FUNCTION_BLOCK FB_SlitPairV2
VAR_INPUT
    nIdPositiveAxis: UINT; //ID of axis for which positive motion increases gap size
    nIdNegativeAxis: UINT; //ID of axis for which negative motion increases gap size
    nIdGapSizeAxis: UINT; //ID of virtual gap aperture size axis
    nIdGapCentreAxis: UINT; //ID of virtual gap centre position axis

    bEnable: BOOL; //Enable slit pair logic functionality
    bReset: BOOL; //Reset from error state
    fEncoderScaling: LREAL := 10000; //Virtual axis scaling denominator, default of 10000
END_VAR
VAR
    nGapSizeEncoder AT %Q*: UDINT := 0;
    nGapCentreEncoder AT %Q*: UDINT := 0;
    fGapSize: LREAL;
    fGapCentre: LREAL;
    bAllHalted: BOOL := FALSE;
    bInternalResetHome: BOOL :=FALSE;

    fbSetpointGenEnablePositiveAxis: MC_ExtSetPointGenEnable;
    fbSetpointGenEnableNegativeAxis: MC_ExtSetPointGenEnable;
    fbSetpointGenEnableGapSizeAxis: MC_ExtSetPointGenEnable;
    fbSetpointGenEnableGapCentreAxis: MC_ExtSetPointGenEnable;

    fbSetpointGenDisablePositiveAxis: MC_ExtSetPointGenDisable;
    fbSetpointGenDisableNegativeAxis: MC_ExtSetPointGenDisable;
    fbSetpointGenDisableGapSizeAxis: MC_ExtSetPointGenDisable;
    fbSetpointGenDisableGapCentreAxis: MC_ExtSetPointGenDisable;

    fPosSetpointPositiveAxis: LREAL;
    fPosSetpointNegativeAxis: LREAL;
    fPosSetpointGapSizeAxis: LREAL;
    fPosSetpointGapCentreAxis: LREAL;

    fVeloSetpointPositiveAxis: LREAL;
    fVeloSetpointNegativeAxis: LREAL;
    fVeloSetpointGapSizeAxis: LREAL;
    fVeloSetpointGapCentreAxis: LREAL;

    nDirectionPositiveAxis: DINT;
    nDirectionNegativeAxis: DINT;
    nDirectionGapSizeAxis: DINT;
    nDirectionGapCentreAxis: DINT;

    eState: E_SlitPairStatesV2 := E_SlitPairStatesV2.eInit;

    bInternalReset: BOOL;
    bHomingReset: BOOL := FALSE;

    //Two resets required due to homing functionality
    bResetInProgressCheck1: BOOL := FALSE;
    bResetInProgressCheck2: BOOL := FALSE;

    //internal MCPOWER blocks because Beckhoff won't let you enable a setpoint generator on a limit....
    fbPowerPositiveAxis: MC_POWER;
    fbPowerNegativeAxis: MC_POWER;
    fbPowerGapSizeAxis: MC_POWER;
    fbPowerGapCentreAxis: MC_POWER;

    //internal MC_Reset, needed because the current reset in FB_Axis works only when there is an error. This should change once the reset functionality changes
    fbInternalResetTrig: R_TRIG;
    fbInternalResetHome: R_TRIG;
    fbResetPositiveAxis: MC_RESET;
    fbResetNegativeAxis: MC_RESET;
    fbResetGapSizeAxis: MC_RESET;
    fbResetGapCentreAxis: MC_RESET;
    fbResetHomedGap: MC_Home;
    fbResetHomedCentre: MC_Home;

END_VAR


(*SETUP INSTRUCTIONS
Virtual axes:
Encoder type set to Universal
Encoder mask set to 0xFFFFFFFF
Encoder scaling set to match FB
Link nDataIn1 of encoder to FB encoders
Position lag monitoring can be left on*
Dynamics of virtual axes must be configured considering coupled mechanicals (e.g. don't set velocities your real axes can't achieve)
*)

//Position of virtual axes
actVirtualAxisPositions();
//Limit logic
actVirtualAxisLimits();
//Enable Logic - Virtual axes automatically enable when real axes are enabled
actVirtualAxisEnable();
//Call spGenerator FBs
actGeneratorEnableDisable();
//Calculate position setpoints
actCalculateSetpointPositions();
//Calculate velocity setpoints
actCalculateSetpointVelocities();
//Calculate directions
actCalculateSetpointDirections();

//Error state handling - only handle errors that disable motion
IF bEnable AND (GVL.astAxesLocal[nIdPositiveAxis].Axis.Status.ErrorStop OR GVL.astAxesLocal[nIdNegativeAxis].Axis.Status.ErrorStop OR GVL.astAxesLocal[nIdGapSizeAxis].Axis.Status.ErrorStop OR GVL.astAxesLocal[nIdGapCentreAxis].Axis.Status.ErrorStop) THEN
    eState := E_SlitPairStatesV2.eError;
END_IF

//Propagate real axis error to virtual
IF GVL.astAxesLocal[nIdPositiveAxis].Axis.Status.ErrorStop AND (NOT GVL.astAxesLocal[nIdGapSizeAxis].Axis.Status.ErrorStop OR NOT GVL.astAxesLocal[nIdGapCentreAxis].Axis.Status.ErrorStop) THEN
    GVL.astAxesLocal[nIdGapSizeAxis].stStatus.bError := TRUE;
    GVL.astAxesLocal[nIdGapCentreAxis].stStatus.bError := TRUE;
    GVL.astAxesLocal[nIdGapSizeAxis].stStatus.nErrorID := GVL.astAxesLocal[nIdPositiveAxis].stStatus.nErrorID;
    GVL.astAxesLocal[nIdGapCentreAxis].stStatus.nErrorID := GVL.astAxesLocal[nIdPositiveAxis].stStatus.nErrorID;
ELSIF  GVL.astAxesLocal[nIdNegativeAxis].Axis.Status.ErrorStop AND (NOT GVL.astAxesLocal[nIdGapSizeAxis].Axis.Status.ErrorStop OR NOT GVL.astAxesLocal[nIdGapCentreAxis].Axis.Status.ErrorStop) THEN
    GVL.astAxesLocal[nIdGapSizeAxis].stStatus.bError := TRUE;
    GVL.astAxesLocal[nIdGapCentreAxis].stStatus.bError := TRUE;
    GVL.astAxesLocal[nIdGapSizeAxis].stStatus.nErrorID := GVL.astAxesLocal[nIdNegativeAxis].stStatus.nErrorID;
    GVL.astAxesLocal[nIdGapCentreAxis].stStatus.nErrorID := GVL.astAxesLocal[nIdNegativeAxis].stStatus.nErrorID;
END_IF

//Internal Reset linked to any axis reset
bInternalReset := bReset OR GVL.astAxesLocal[nIdPositiveAxis].stControl.bReset OR GVL.astAxesLocal[nIdNegativeAxis].stControl.bReset OR GVL.astAxesLocal[nIdGapSizeAxis].stControl.bReset OR GVL.astAxesLocal[nIdGapCentreAxis].stControl.bReset;

//If real axis is homing, change state
IF bEnable AND (GVL.astAxesLocal[nIdPositiveAxis].Axis.Status.HomingBusy OR GVL.astAxesLocal[nIdNegativeAxis].Axis.Status.HomingBusy) THEN
    eState := E_SlitPairStatesV2.eWaitForRealHomed;
END_IF

//Link all halt buttons in motors
IF GVL.astAxesLocal[nIdPositiveAxis].stControl.bHalt OR GVL.astAxesLocal[nIdNegativeAxis].stControl.bHalt OR
    GVL.astAxesLocal[nIdGapSizeAxis].stControl.bHalt OR GVL.astAxesLocal[nIdGapCentreAxis].stControl.bHalt THEN
    actHaltAllAxes();
END_IF

//Propagate homing status
fbResetHomedGap(Axis:= GVL.astAxesLocal[nIdGapSizeAxis].Axis, HomingMode:= MC_ResetCalibration);
fbResetHomedCentre(Axis:= GVL.astAxesLocal[nIdGapCentreAxis].Axis, HomingMode:= MC_ResetCalibration);
fbInternalResetHome(CLK:= fbResetHomedCentre.Done OR fbResetHomedGap.Done );
IF NOT GVL.astAxesLocal[nIdPositiveAxis].stStatus.bHomed OR NOT GVL.astAxesLocal[nIdNegativeAxis].stStatus.bHomed THEN
        fbResetHomedGap.Execute := TRUE;
        fbResetHomedCentre.Execute := TRUE;
END_IF

IF fbInternalResetHome.Q THEN
        fbResetHomedGap.Execute := FALSE;
        fbResetHomedCentre.Execute := FALSE;
END_IF


//State machine
IF bEnable THEN
    CASE eState OF  //HOMING LOOP ISSUE
        E_SlitPairStatesV2.eInit:
            //If real axes are calibrated, then home the virtual axes, else go Operatioanl
            fbResetPositiveAxis(Axis:=GVL.astAxesLocal[nIdPositiveAxis].Axis, Execute:=FALSE);
            fbResetNegativeAxis(Axis:=GVL.astAxesLocal[nIdNegativeAxis].Axis, Execute:=FALSE);
            fbResetGapSizeAxis(Axis:=GVL.astAxesLocal[nIdGapSizeAxis].Axis, Execute:=FALSE);
            fbResetGapCentreAxis(Axis:=GVL.astAxesLocal[nIdGapCentreAxis].Axis, Execute:=FALSE);
            IF GVL.astAxesLocal[nIdPositiveAxis].stStatus.bHomed AND GVL.astAxesLocal[nIdNegativeAxis].stStatus.bHomed THEN
               GVL.astAxesLocal[nIdGapSizeAxis].stConfig.eHomeSeq := E_HomingRoutines.eHomeDirect;
               GVL.astAxesLocal[nIdGapCentreAxis].stConfig.eHomeSeq := E_HomingRoutines.eHomeDirect;
               GVL.astAxesLocal[nIdGapSizeAxis].stConfig.fHomePosition := fGapSize;
               GVL.astAxesLocal[nIdGapCentreAxis].stConfig.fHomePosition := fGapCentre;
                eState := E_SlitPairStatesV2.eWaitForVirtualHomed;
            ELSE
                eState := E_SlitPairStatesV2.eOperational;
            END_IF

        E_SlitPairStatesV2.eWaitForVirtualHomed:
            //Wait for virtual axis homing to complete/
            GVL.astAxesLocal[nIdGapSizeAxis].stControl.eCommand := E_MotionFunctions.eHome;
            GVL.astAxesLocal[nIdGapSizeAxis].stControl.bExecute := TRUE;
            GVL.astAxesLocal[nIdGapCentreAxis].stControl.eCommand := E_MotionFunctions.eHome;
            GVL.astAxesLocal[nIdGapCentreAxis].stControl.bExecute := TRUE;
            IF GVL.astAxesLocal[nIdGapSizeAxis].stStatus.bHomed AND GVL.astAxesLocal[nIdGapCentreAxis].stStatus.bHomed THEN
                eState := E_SlitPairStatesV2.eOperational;
            END_IF
            //IF NOT IN HOMING STATE

        E_SlitPairStatesV2.eOperational:
            bResetInProgressCheck1 := FALSE;
            //Detect whether real or virtual axes are moving
            IF GVL.astAxesLocal[nIdGapSizeAxis].stStatus.bMoving OR GVL.astAxesLocal[nIdGapCentreAxis].stStatus.bMoving THEN
                eState := E_SlitPairStatesV2.eEnableRealGenerators;
            END_IF
            IF GVL.astAxesLocal[nIdPositiveAxis].stStatus.bMoving OR GVL.astAxesLocal[nIdNegativeAxis].stStatus.bMoving THEN
                eState := E_SlitPairStatesV2.eEnableVirtualGenerators;
            END_IF

        E_SlitPairStatesV2.eEnableRealGenerators:
            //Hold MC_Power on until generators have enabled
            fbPowerPositiveAxis(Axis:=GVL.astAxesLocal[nIdPositiveAxis].Axis, Enable:=TRUE, Enable_Positive:=TRUE,Enable_Negative:=TRUE);
            fbPowerNegativeAxis(Axis:=GVL.astAxesLocal[nIdNegativeAxis].Axis, Enable:=TRUE, Enable_Positive:=TRUE,Enable_Negative:=TRUE);
            fbSetpointGenEnablePositiveAxis.Execute := TRUE;
            fbSetpointGenEnableNegativeAxis.Execute := TRUE;
            eState := E_SlitPairStatesV2.eCheckRealAxisGeneratorsEnabled;

        E_SlitPairStatesV2.eCheckRealAxisGeneratorsEnabled:
            //Hold MC_Power on until generators have enabled
            fbPowerPositiveAxis(Axis:=GVL.astAxesLocal[nIdPositiveAxis].Axis, Enable:=TRUE, Enable_Positive:=TRUE,Enable_Negative:=TRUE);
            fbPowerNegativeAxis(Axis:=GVL.astAxesLocal[nIdNegativeAxis].Axis, Enable:=TRUE, Enable_Positive:=TRUE,Enable_Negative:=TRUE);
            IF fbSetpointGenEnablePositiveAxis.Enabled AND fbSetpointGenEnableNegativeAxis.Enabled THEN
                eState := E_SlitPairStatesV2.eWaitForVirtualMoveDone;
            END_IF

        E_SlitPairStatesV2.eWaitForVirtualMoveDone:
            IF NOT(GVL.astAxesLocal[nIdGapSizeAxis].stStatus.bMoving OR GVL.astAxesLocal[nIdGapCentreAxis].stStatus.bMoving) THEN
                eState := E_SlitPairStatesV2.eDisableRealGenerators;
            END_IF

        E_SlitPairStatesV2.eDisableRealGenerators:
            fbSetpointGenDisablePositiveAxis.Execute := TRUE;
            fbSetpointGenDisableNegativeAxis.Execute := TRUE;
            eState := E_SlitPairStatesV2.eOperational;

        E_SlitPairStatesV2.eEnableVirtualGenerators:
            //Hold MC_Power on until generators have enabled
            fbPowerGapSizeAxis(Axis:=GVL.astAxesLocal[nIdGapSizeAxis].Axis, Enable:=TRUE, Enable_Positive:=TRUE,Enable_Negative:=TRUE);
            fbPowerGapCentreAxis(Axis:=GVL.astAxesLocal[nIdGapCentreAxis].Axis, Enable:=TRUE, Enable_Positive:=TRUE,Enable_Negative:=TRUE);
            fbSetpointGenEnableGapSizeAxis.Execute := TRUE;
            fbSetpointGenEnableGapCentreAxis.Execute := TRUE;
            eState := E_SlitPairStatesV2.eCheckVirtualAxisGeneratorsEnabled;

        E_SlitPairStatesV2.eCheckVirtualAxisGeneratorsEnabled:
            //Hold MC_Power on until generators have enabled
            fbPowerGapSizeAxis(Axis:=GVL.astAxesLocal[nIdGapSizeAxis].Axis, Enable:=TRUE, Enable_Positive:=TRUE,Enable_Negative:=TRUE);
            fbPowerGapCentreAxis(Axis:=GVL.astAxesLocal[nIdGapCentreAxis].Axis, Enable:=TRUE, Enable_Positive:=TRUE,Enable_Negative:=TRUE);
            IF fbSetpointGenEnableGapSizeAxis.Enabled AND fbSetpointGenEnableGapCentreAxis.Enabled THEN
                eState := E_SlitPairStatesV2.eWaitForRealMoveDone;
            END_IF

        E_SlitPairStatesV2.eWaitForRealMoveDone:
            IF NOT(GVL.astAxesLocal[nIdPositiveAxis].stStatus.bMoving OR GVL.astAxesLocal[nIdNegativeAxis].stStatus.bMoving) THEN
                eState := E_SlitPairStatesV2.eDisableVirtualGenerators;
            END_IF

        E_SlitPairStatesV2.eDisableVirtualGenerators:
            fbSetpointGenDisableGapSizeAxis.Execute := TRUE;
            fbSetpointGenDisableGapCentreAxis.Execute := TRUE;
            eState := E_SlitPairStatesV2.eOperational;

        E_SlitPairStatesV2.eError:
            actHaltAllAxes();

            IF bHomingReset THEN
                bInternalReset := TRUE;
                bResetInProgressCheck1 := TRUE;
                bResetInProgressCheck2 := TRUE;
                bHomingReset := FALSE;
            END_IF
            IF bInternalReset OR bReset OR bResetInProgressCheck2 THEN
                fbResetPositiveAxis(Axis:=GVL.astAxesLocal[nIdPositiveAxis].Axis, Execute:=TRUE);
                fbResetNegativeAxis(Axis:=GVL.astAxesLocal[nIdNegativeAxis].Axis, Execute:=TRUE);
                fbResetGapSizeAxis(Axis:=GVL.astAxesLocal[nIdGapSizeAxis].Axis, Execute:=TRUE);
                fbResetGapCentreAxis(Axis:=GVL.astAxesLocal[nIdGapCentreAxis].Axis, Execute:=TRUE);
                GVL.astAxesLocal[nIdPositiveAxis].stControl.bReset := TRUE;
                GVL.astAxesLocal[nIdNegativeAxis].stControl.bReset := TRUE;
                GVL.astAxesLocal[nIdGapSizeAxis].stControl.bReset := TRUE;
                GVL.astAxesLocal[nIdGapCentreAxis].stControl.bReset := TRUE;
                IF NOT(bResetInProgressCheck1) THEN
                    bResetInProgressCheck2 := FALSE;
                END_IF
            END_IF

            IF NOT(GVL.astAxesLocal[nIdPositiveAxis].stStatus.bError) AND NOT(GVL.astAxesLocal[nIdNegativeAxis].stStatus.bError) AND NOT(GVL.astAxesLocal[nIdGapSizeAxis].stStatus.bError) AND NOT(GVL.astAxesLocal[nIdGapCentreAxis].stStatus.bError) THEN
                eState := E_SlitPairStatesV2.eInit;
            END_IF

        E_SlitPairStatesV2.eWaitForRealHomed:
            bHomingReset := TRUE;
            IF NOT GVL.astAxesLocal[nIdPositiveAxis].Axis.Status.Homed OR NOT GVL.astAxesLocal[nIdNegativeAxis].Axis.Status.Homed THEN
                eState := E_SlitPairStatesV2.eInit;
            END_IF
    END_CASE
END_IF


//Feed externalsetpoint generators setpoint values - ignoring acceleration
MC_ExtSetPointGenFeed(Axis:= GVL.astAxesLocal[nIdPositiveAxis].Axis, Position:= fPosSetpointPositiveAxis, Velocity:= fVeloSetpointPositiveAxis, Acceleration:= 0, Direction:= nDirectionPositiveAxis);
MC_ExtSetPointGenFeed(Axis:= GVL.astAxesLocal[nIdNegativeAxis].Axis, Position:= fPosSetpointNegativeAxis, Velocity:= fVeloSetpointNegativeAxis, Acceleration:= 0, Direction:= nDirectionNegativeAxis);
MC_ExtSetPointGenFeed(Axis:= GVL.astAxesLocal[nIdGapSizeAxis].Axis, Position:= fPosSetpointGapSizeAxis, Velocity:= fVeloSetpointGapSizeAxis, Acceleration:= 0, Direction:= nDirectionGapSizeAxis);
MC_ExtSetPointGenFeed(Axis:= GVL.astAxesLocal[nIdGapCentreAxis].Axis, Position:= fPosSetpointGapCentreAxis, Velocity:= fVeloSetpointGapCentreAxis, Acceleration:= 0, Direction:= nDirectionGapCentreAxis);

bReset := FALSE;

ACTION actCalculateSetpointDirections:

IF fVeloSetpointPositiveAxis > 0 THEN
    nDirectionPositiveAxis := 1; //moving forward
ELSIF fVeloSetpointPositiveAxis < 0 THEN
    nDirectionPositiveAxis := -1; //moving backward
ELSE
    nDirectionPositiveAxis := 0; //stationary
END_IF

IF fVeloSetpointNegativeAxis > 0 THEN
    nDirectionNegativeAxis := 1; //moving forward
ELSIF fVeloSetpointNegativeAxis < 0 THEN
    nDirectionNegativeAxis := -1; //moving backward
ELSE
    nDirectionNegativeAxis := 0; //stationary
END_IF

IF fVeloSetpointGapSizeAxis > 0 THEN
    nDirectionGapSizeAxis := 1; //moving forward
ELSIF fVeloSetpointGapSizeAxis < 0 THEN
    nDirectionGapSizeAxis := -1; //moving backward
ELSE
    nDirectionGapSizeAxis := 0; //stationary
END_IF

IF fVeloSetpointGapCentreAxis > 0 THEN
    nDirectionGapCentreAxis := 1; //moving forward
ELSIF fVeloSetpointGapCentreAxis < 0 THEN
    nDirectionGapCentreAxis := -1; //moving backward
ELSE
    nDirectionGapCentreAxis := 0; //stationary
END_IF
END_ACTION

ACTION actCalculateSetpointPositions:

fPosSetpointPositiveAxis := GVL.astAxesLocal[nIdGapCentreAxis].Axis.NcToPlc.SetPos + (GVL.astAxesLocal[nIdGapSizeAxis].Axis.NcToPlc.SetPos/2);
fPosSetpointNegativeAxis := GVL.astAxesLocal[nIdGapCentreAxis].Axis.NcToPlc.SetPos - (GVL.astAxesLocal[nIdGapSizeAxis].Axis.NcToPlc.SetPos/2);
fPosSetpointGapSizeAxis := GVL.astAxesLocal[nIdPositiveAxis].Axis.NcToPlc.SetPos - GVL.astAxesLocal[nIdNegativeAxis].Axis.NcToPlc.SetPos;
fPosSetpointGapCentreAxis := (GVL.astAxesLocal[nIdPositiveAxis].Axis.NcToPlc.SetPos + GVL.astAxesLocal[nIdNegativeAxis].Axis.NcToPlc.SetPos) / 2;
END_ACTION

ACTION actCalculateSetpointVelocities:

fVeloSetpointPositiveAxis := GVL.astAxesLocal[nIdGapCentreAxis].Axis.NcToPlc.SetVelo +(GVL.astAxesLocal[nIdGapSizeAxis].Axis.NcToPlc.SetVelo/2);
fVeloSetpointNegativeAxis := GVL.astAxesLocal[nIdGapCentreAxis].Axis.NcToPlc.SetVelo -(GVL.astAxesLocal[nIdGapSizeAxis].Axis.NcToPlc.SetVelo/2);
fVeloSetpointGapSizeAxis := GVL.astAxesLocal[nIdPositiveAxis].Axis.NcToPlc.SetVelo - GVL.astAxesLocal[nIdNegativeAxis].Axis.NcToPlc.SetVelo;
fVeloSetpointGapCentreAxis := GVL.astAxesLocal[nIdPositiveAxis].Axis.NcToPlc.SetVelo + GVL.astAxesLocal[nIdNegativeAxis].Axis.NcToPlc.SetVelo;
END_ACTION

ACTION actGeneratorEnableDisable:

fbSetpointGenEnablePositiveAxis(Axis:=GVL.astAxesLocal[nIdPositiveAxis].Axis);
fbSetpointGenEnablePositiveAxis.Execute := FALSE;

fbSetpointGenEnableNegativeAxis(Axis:=GVL.astAxesLocal[nIdNegativeAxis].Axis);
fbSetpointGenEnableNegativeAxis.Execute := FALSE;

fbSetpointGenEnableGapSizeAxis(Axis:=GVL.astAxesLocal[nIdGapSizeAxis].Axis);
fbSetpointGenEnableGapSizeAxis.Execute := FALSE;

fbSetpointGenEnableGapCentreAxis(Axis:=GVL.astAxesLocal[nIdGapCentreAxis].Axis);
fbSetpointGenEnableGapCentreAxis.Execute := FALSE;


fbSetpointGenDisablePositiveAxis(Axis:=GVL.astAxesLocal[nIdPositiveAxis].Axis);
fbSetpointGenDisablePositiveAxis.Execute := FALSE;

fbSetpointGenDisableNegativeAxis(Axis:=GVL.astAxesLocal[nIdNegativeAxis].Axis);
fbSetpointGenDisableNegativeAxis.Execute := FALSE;

fbSetpointGenDisableGapSizeAxis(Axis:=GVL.astAxesLocal[nIdGapSizeAxis].Axis);
fbSetpointGenDisableGapSizeAxis.Execute := FALSE;

fbSetpointGenDisableGapCentreAxis(Axis:=GVL.astAxesLocal[nIdGapCentreAxis].Axis);
fbSetpointGenDisableGapCentreAxis.Execute := FALSE;
END_ACTION

ACTION actHaltAllAxes:

GVL.astAxesLocal[nIdPositiveAxis].stControl.bHalt := TRUE;
GVL.astAxesLocal[nIdNegativeAxis].stControl.bHalt := TRUE;
GVL.astAxesLocal[nIdGapSizeAxis].stControl.bHalt := TRUE;
GVL.astAxesLocal[nIdGapCentreAxis].stControl.bHalt := TRUE;
bAllHalted := TRUE;

//Reset Halts
IF bAllHalted AND NOT GVL.astAxesLocal[nIdPositiveAxis].stStatus.bMoving AND NOT GVL.astAxesLocal[nIdNegativeAxis].stStatus.bMoving
 AND NOT GVL.astAxesLocal[nIdGapSizeAxis].stStatus.bMoving AND NOT GVL.astAxesLocal[nIdGapCentreAxis].stStatus.bMoving THEN
   GVL.astAxesLocal[nIdPositiveAxis].stControl.bHalt := FALSE;
   GVL.astAxesLocal[nIdNegativeAxis].stControl.bHalt := FALSE;
   GVL.astAxesLocal[nIdGapSizeAxis].stControl.bHalt := FALSE;
   GVL.astAxesLocal[nIdGapCentreAxis].stControl.bHalt := FALSE;
   bAllHalted := FALSE;
END_IF
END_ACTION

ACTION actVirtualAxisEnable:

GVL.astAxesLocal[nIdGapSizeAxis].stControl.bEnable := GVL.astAxesLocal[nIdPositiveAxis].stStatus.bEnabled AND GVL.astAxesLocal[nIdNegativeAxis].stStatus.bEnabled;
GVL.astAxesLocal[nIdGapCentreAxis].stControl.bEnable := GVL.astAxesLocal[nIdPositiveAxis].stStatus.bEnabled AND GVL.astAxesLocal[nIdNegativeAxis].stStatus.bEnabled;
END_ACTION

ACTION actVirtualAxisLimits:

GVL.astAxesLocal[nIdGapSizeAxis].stInputs.bLimitFwd := GVL.astAxesLocal[nIdPositiveAxis].stStatus.bFwEnabled AND GVL.astAxesLocal[nIdNegativeAxis].stStatus.bBwEnabled;
GVL.astAxesLocal[nIdGapSizeAxis].stInputs.bLimitBwd := GVL.astAxesLocal[nIdPositiveAxis].stStatus.bBwEnabled AND GVL.astAxesLocal[nIdNegativeAxis].stStatus.bFwEnabled;

GVL.astAxesLocal[nIdGapCentreAxis].stInputs.bLimitFwd := GVL.astAxesLocal[nIdPositiveAxis].stStatus.bFwEnabled AND GVL.astAxesLocal[nIdNegativeAxis].stStatus.bFwEnabled;
GVL.astAxesLocal[nIdGapCentreAxis].stInputs.bLimitBwd := GVL.astAxesLocal[nIdPositiveAxis].stStatus.bBwEnabled AND GVL.astAxesLocal[nIdNegativeAxis].stStatus.bBwEnabled;
END_ACTION

ACTION actVirtualAxisPositions:

(*Calculate virtual axis positions and convert to UDINT.
Conversion to UDINT is prohibited if it would exceed UDINT max value of 4,294,967,295.
If this is not done, it can cause overflow when connected to the encoder input and hard-crash the PLC which will only recover with a power cycle.
To preserve decimal position data of the LREAL (i.e. anything <1mm) it is necessary to scale the value before converting to UDINT.
This can be reversed with the correct scaling at the NC encoder level.
*)
fGapSize := GVL.astAxesLocal[nIdPositiveAxis].stStatus.fActPosition - GVL.astAxesLocal[nIdNegativeAxis].stStatus.fActPosition;
fGapCentre := (GVL.astAxesLocal[nIdPositiveAxis].stStatus.fActPosition + GVL.astAxesLocal[nIdNegativeAxis].stStatus.fActPosition)/2;


    IF ABS(fGapSize) < 100000 THEN
        nGapSizeEncoder := LREAL_TO_UDINT(fGapSize*fEncoderScaling);
    END_IF
    IF ABS(fGapCentre) < 100000 THEN
        nGapCentreEncoder := LREAL_TO_UDINT(fGapCentre*fEncoderScaling);
    END_IF
END_ACTION

END_FUNCTION_BLOCK

(* stored: Version 1.1.0.1, ProductVersion 3.1.4026.18
   POU FB_SlitPairV2: Id {ff4013b1-472a-4f42-a6c8-2711712ac06d}, SpecialFunc None
   Action actCalculateSetpointDirections: Id {7783e346-7fab-40d5-bab7-fe46a8c2f785}
   Action actCalculateSetpointPositions: Id {08e35b97-914a-4ccc-a3af-6b7cd8e60439}
   Action actCalculateSetpointVelocities: Id {59813eea-6905-4661-a8f3-10b16a472979}
   Action actGeneratorEnableDisable: Id {d59f6d39-50eb-4cb0-8d9d-b62df150c5a5}
   Action actHaltAllAxes: Id {f2afb93d-4a80-499a-b8ec-4e673220e7ad}
   Action actVirtualAxisEnable: Id {d8729d12-361d-472b-8974-5b566dad7d06}
   Action actVirtualAxisLimits: Id {436d835a-8846-47e9-922d-a1df63469a25}
   Action actVirtualAxisPositions: Id {4ef557a2-3171-4a03-98ba-14f2cd3ef5ec} *)
